// TIA Portal V18 export
DATA_BLOCK "L1_lubrificazioni"   // DB11
{ S7_Optimized_Access := 'TRUE' }
VERSION : 0.1
// stored: AutoNumber true, DBAccessibleFromOPCUA true, DBAccessibleFromWebserver true, IsOnlyStoredInLoadMemory false, IsRetainMemResEnabled false, IsWriteProtectedInAS false, MemoryReserve 100
   VAR RETAIN
      num { S7_SetPoint := 'True'} : Array[1..10] of "LGasp_type_lubrificazioniPC";
   END_VAR
BEGIN
   num[1..10].tipo := 0;
   num[1].nome := WSTRING#'prova';
   num[2..10].nome := WSTRING#'';
   num[1].nometrad := WSTRING#'Lub.Lamiera';
   num[2..10].nometrad := WSTRING#'';
   num[1..10].cmdabilitata := FALSE;
   num[1..10].cmdmanuale := FALSE;
   num[1..10].cmddurata := 0.0;
   num[1..10].cmdquota := 0.0;
   num[1..10].stsquotaattuale := 0.0;
   num[1..10].cmdnumcolpi := 0.0;
   num[1..10].stsnumcolpiattuali := 0.0;
   num[1..10].cmdritardo := 0.0;
   num[1..10].stsRitardoattuale := 0.0;
END_DATA_BLOCK
